// TIA Portal V17 export
// export: Created 2024-09-02T12:50:19.8771869Z, ExportSetting WithDefaults, DisplayName Totally Integrated Automation Portal, DisplayVersion V17, DisplayName TIA Portal Openness, DisplayVersion V17, DisplayName TIA Portal Version Control Interface, DisplayVersion V17, DisplayName STEP 7 Professional, DisplayVersion V17, DisplayName STEP 7 Safety, DisplayVersion V17, DisplayName WinCC Professional, DisplayVersion V17
FUNCTION "AnwFC1_FG02_Parameter_SLG3_OP70" : Void   // FC1111, LAD
TITLE = Parameter Moby / Parameter Moby
{ S7_Optimized_Access := 'TRUE' }
AUTHOR : OlegFuehrus
FAMILY : MOBY
NAME : OlegFuehrus
VERSION : 0.1
// stored: AutoNumber false, IsIECCheckEnabled false, SetENOAutomatically false, UDAEnableTagReadback false
   VAR_TEMP
      Motion_Release : Bool;
      Hand : Bool;
      Auto : Bool;
      t_VKE0 : Bool;
      t_VKE1 : Bool;
      t_reset : Bool;
      t_read : Bool;
      t_read_ok : Bool;
      t_write : Bool;
      t_write_ok : Bool;
      t_TAFmaske : Byte;
      t_PageNr_Station : Int;
      t_PageNr_Station_Before : Int;
      t_Nr : Int;
      Length_of_Db : Int;
   END_VAR
   VAR_TEMP   // added for the SCL form of the ladder/FBD networks
      _w1 : Bool;
   END_VAR
BEGIN

REGION Network 1: VKE 0/1
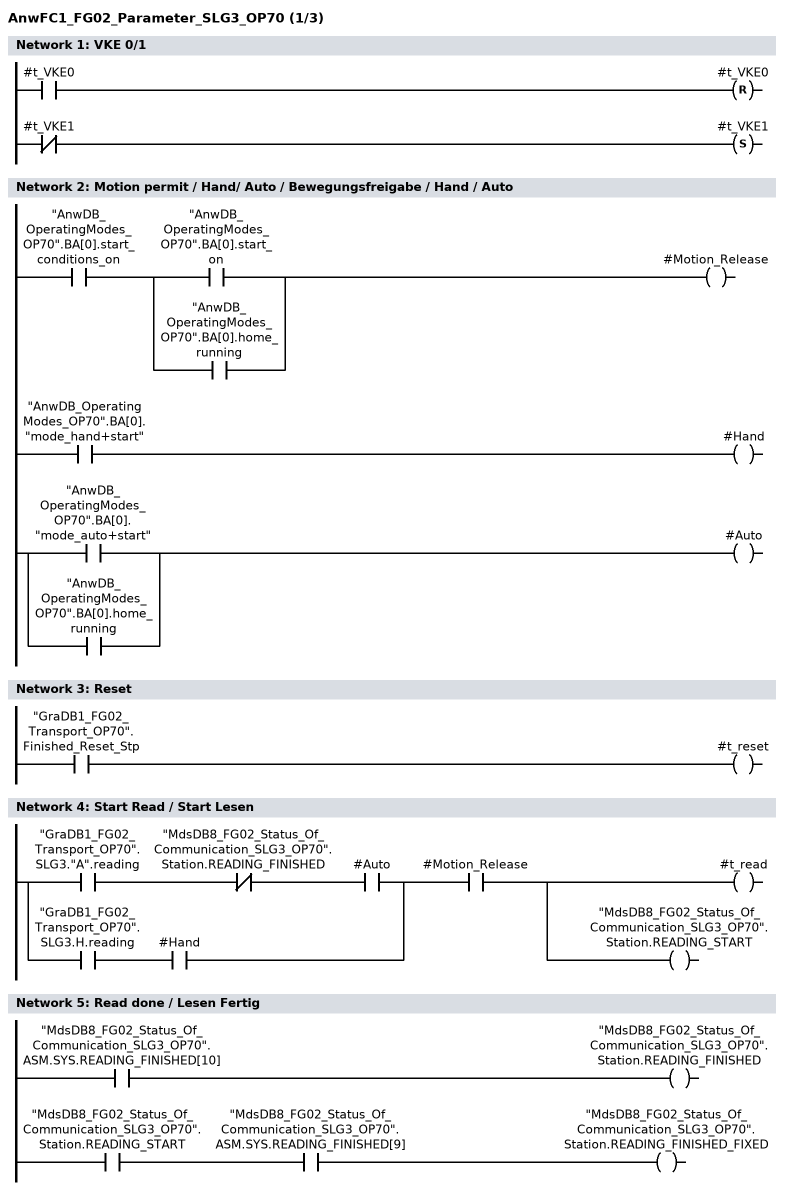
   RUNG wire#powerrail
      Contact( #t_VKE0 )
      R_Coil( #t_VKE0 )
   END_RUNG
   RUNG wire#powerrail
      I_Contact( #t_VKE1 )
      S_Coil( #t_VKE1 )
   END_RUNG
   // the same network as SCL:
   IF #t_VKE0 THEN #t_VKE0 := FALSE; END_IF;
   IF NOT #t_VKE1 THEN #t_VKE1 := TRUE; END_IF;
END_REGION

REGION Network 2: Motion permit / Hand/ Auto / Bewegungsfreigabe / Hand / Auto
   RUNG wire#powerrail
      Contact( "AnwDB_OperatingModes_OP70".BA[0].start_conditions_on )
      wire#w1
      Contact( "AnwDB_OperatingModes_OP70".BA[0].start_on )
      wire#w2
      Coil( #Motion_Release )
   END_RUNG
   RUNG wire#w1
      Contact( "AnwDB_OperatingModes_OP70".BA[0].home_running )
   END_RUNG wire#w2
   RUNG wire#powerrail
      Contact( "AnwDB_OperatingModes_OP70".BA[0]."mode_hand+start" )
      Coil( #Hand )
   END_RUNG
   RUNG wire#powerrail
      Contact( "AnwDB_OperatingModes_OP70".BA[0]."mode_auto+start" )
      wire#w3
      Coil( #Auto )
   END_RUNG
   RUNG wire#powerrail
      Contact( "AnwDB_OperatingModes_OP70".BA[0].home_running )
   END_RUNG wire#w3
   // the same network as SCL:
   #Motion_Release := "AnwDB_OperatingModes_OP70".BA[0].start_conditions_on AND ("AnwDB_OperatingModes_OP70".BA[0].start_on OR "AnwDB_OperatingModes_OP70".BA[0].home_running);
   #Hand := "AnwDB_OperatingModes_OP70".BA[0]."mode_hand+start";
   #Auto := "AnwDB_OperatingModes_OP70".BA[0]."mode_auto+start" OR "AnwDB_OperatingModes_OP70".BA[0].home_running;
END_REGION

REGION Network 3: Reset
   RUNG wire#powerrail
      Contact( "GraDB1_FG02_Transport_OP70".Finished_Reset_Stp )
      Coil( #t_reset )
   END_RUNG
   // the same network as SCL:
   #t_reset := "GraDB1_FG02_Transport_OP70".Finished_Reset_Stp;
END_REGION

REGION Network 4: Start Read / Start Lesen
   RUNG wire#powerrail
      Contact( "GraDB1_FG02_Transport_OP70".SLG3."A".reading )
      I_Contact( "MdsDB8_FG02_Status_Of_Communication_SLG3_OP70".Station.READING_FINISHED )
      Contact( #Auto )
      wire#w1
      Contact( #Motion_Release )
      wire#w2
      Coil( #t_read )
   END_RUNG
   RUNG wire#powerrail
      Contact( "GraDB1_FG02_Transport_OP70".SLG3.H.reading )
      Contact( #Hand )
   END_RUNG wire#w1
   RUNG wire#w2
      Coil( "MdsDB8_FG02_Status_Of_Communication_SLG3_OP70".Station.READING_START )
   END_RUNG
   // the same network as SCL:
   #t_read := (("GraDB1_FG02_Transport_OP70".SLG3."A".reading AND NOT "MdsDB8_FG02_Status_Of_Communication_SLG3_OP70".Station.READING_FINISHED AND #Auto) OR ("GraDB1_FG02_Transport_OP70".SLG3.H.reading AND #Hand)) AND #Motion_Release;
   "MdsDB8_FG02_Status_Of_Communication_SLG3_OP70".Station.READING_START := #t_read;
END_REGION

REGION Network 5: Read done / Lesen Fertig
   RUNG wire#powerrail
      Contact( "MdsDB8_FG02_Status_Of_Communication_SLG3_OP70".ASM.SYS.READING_FINISHED[10] )
      Coil( "MdsDB8_FG02_Status_Of_Communication_SLG3_OP70".Station.READING_FINISHED )
   END_RUNG
   RUNG wire#powerrail
      Contact( "MdsDB8_FG02_Status_Of_Communication_SLG3_OP70".Station.READING_START )
      Contact( "MdsDB8_FG02_Status_Of_Communication_SLG3_OP70".ASM.SYS.READING_FINISHED[9] )
      Coil( "MdsDB8_FG02_Status_Of_Communication_SLG3_OP70".Station.READING_FINISHED_FIXED )
   END_RUNG
   // the same network as SCL:
   "MdsDB8_FG02_Status_Of_Communication_SLG3_OP70".Station.READING_FINISHED := "MdsDB8_FG02_Status_Of_Communication_SLG3_OP70".ASM.SYS.READING_FINISHED[10];
   "MdsDB8_FG02_Status_Of_Communication_SLG3_OP70".Station.READING_FINISHED_FIXED := "MdsDB8_FG02_Status_Of_Communication_SLG3_OP70".Station.READING_START AND "MdsDB8_FG02_Status_Of_Communication_SLG3_OP70".ASM.SYS.READING_FINISHED[9];
END_REGION

REGION Network 6: Start Writing / Start Schreiben
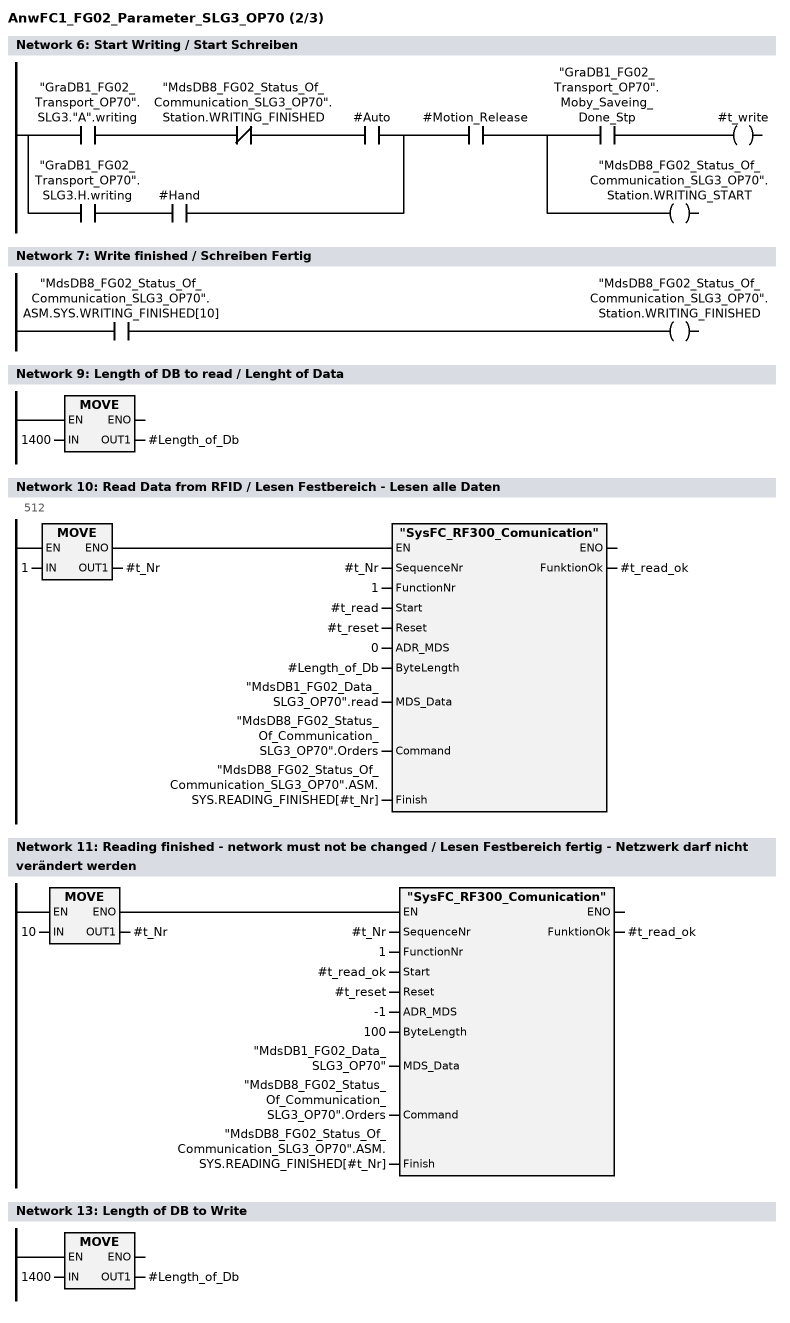
   RUNG wire#powerrail
      Contact( "GraDB1_FG02_Transport_OP70".SLG3."A".writing )
      I_Contact( "MdsDB8_FG02_Status_Of_Communication_SLG3_OP70".Station.WRITING_FINISHED )
      Contact( #Auto )
      wire#w1
      Contact( #Motion_Release )
      wire#w2
      Contact( "GraDB1_FG02_Transport_OP70".Moby_Saveing_Done_Stp )
      Coil( #t_write )
   END_RUNG
   RUNG wire#powerrail
      Contact( "GraDB1_FG02_Transport_OP70".SLG3.H.writing )
      Contact( #Hand )
   END_RUNG wire#w1
   RUNG wire#w2
      Coil( "MdsDB8_FG02_Status_Of_Communication_SLG3_OP70".Station.WRITING_START )
   END_RUNG
   // the same network as SCL:
   #_w1 := (("GraDB1_FG02_Transport_OP70".SLG3."A".writing AND NOT "MdsDB8_FG02_Status_Of_Communication_SLG3_OP70".Station.WRITING_FINISHED AND #Auto) OR ("GraDB1_FG02_Transport_OP70".SLG3.H.writing AND #Hand)) AND #Motion_Release;
   #t_write := #_w1 AND "GraDB1_FG02_Transport_OP70".Moby_Saveing_Done_Stp;
   "MdsDB8_FG02_Status_Of_Communication_SLG3_OP70".Station.WRITING_START := #_w1;
END_REGION

REGION Network 7: Write finished / Schreiben Fertig
   RUNG wire#powerrail
      Contact( "MdsDB8_FG02_Status_Of_Communication_SLG3_OP70".ASM.SYS.WRITING_FINISHED[10] )
      Coil( "MdsDB8_FG02_Status_Of_Communication_SLG3_OP70".Station.WRITING_FINISHED )
   END_RUNG
   // the same network as SCL:
   "MdsDB8_FG02_Status_Of_Communication_SLG3_OP70".Station.WRITING_FINISHED := "MdsDB8_FG02_Status_Of_Communication_SLG3_OP70".ASM.SYS.WRITING_FINISHED[10];
END_REGION

REGION Network 8: ######## READ PARAMETER ########
END_REGION

REGION Network 9: Length of DB to read / Lenght of Data
   RUNG wire#powerrail
      Move(in := 1400, out1 => #Length_of_Db)
   END_RUNG
   // the same network as SCL:
   #Length_of_Db := 1400;
END_REGION

REGION Network 10: Read Data from RFID / Lesen Festbereich - Lesen alle Daten
   // 512
   RUNG wire#powerrail
      Move(in := 1, out1 => #t_Nr)
      "SysFC_RF300_Comunication"(SequenceNr := #t_Nr, FunctionNr := 1, Start := #t_read, Reset := #t_reset, ADR_MDS := 0, ByteLength := #Length_of_Db, MDS_Data := "MdsDB1_FG02_Data_SLG3_OP70".read, Command := "MdsDB8_FG02_Status_Of_Communication_SLG3_OP70".Orders, Finish := "MdsDB8_FG02_Status_Of_Communication_SLG3_OP70".ASM.SYS.READING_FINISHED[#t_Nr], FunktionOk => #t_read_ok)
   END_RUNG
   // the same network as SCL:
   #t_Nr := 1;
   "SysFC_RF300_Comunication"(SequenceNr := #t_Nr,
                           FunctionNr := 1,
                           Start := #t_read,
                           Reset := #t_reset,
                           ADR_MDS := 0,
                           ByteLength := #Length_of_Db,
                           MDS_Data := "MdsDB1_FG02_Data_SLG3_OP70".read,
                           Command := "MdsDB8_FG02_Status_Of_Communication_SLG3_OP70".Orders,
                           Finish := "MdsDB8_FG02_Status_Of_Communication_SLG3_OP70".ASM.SYS.READING_FINISHED[#t_Nr],
                           FunktionOk => #t_read_ok);
END_REGION

REGION Network 11: Reading finished - network must not be changed / Lesen Festbereich fertig - Netzwerk darf nicht verändert werden
   RUNG wire#powerrail
      Move(in := 10, out1 => #t_Nr)
      "SysFC_RF300_Comunication"(SequenceNr := #t_Nr, FunctionNr := 1, Start := #t_read_ok, Reset := #t_reset, ADR_MDS := -1, ByteLength := 100, MDS_Data := "MdsDB1_FG02_Data_SLG3_OP70", Command := "MdsDB8_FG02_Status_Of_Communication_SLG3_OP70".Orders, Finish := "MdsDB8_FG02_Status_Of_Communication_SLG3_OP70".ASM.SYS.READING_FINISHED[#t_Nr], FunktionOk => #t_read_ok)
   END_RUNG
   // the same network as SCL:
   #t_Nr := 10;
   "SysFC_RF300_Comunication"(SequenceNr := #t_Nr,
                           FunctionNr := 1,
                           Start := #t_read_ok,
                           Reset := #t_reset,
                           ADR_MDS := -1,
                           ByteLength := 100,
                           MDS_Data := "MdsDB1_FG02_Data_SLG3_OP70",
                           Command := "MdsDB8_FG02_Status_Of_Communication_SLG3_OP70".Orders,
                           Finish := "MdsDB8_FG02_Status_Of_Communication_SLG3_OP70".ASM.SYS.READING_FINISHED[#t_Nr],
                           FunktionOk => #t_read_ok);
END_REGION

REGION Network 12: ######## WRITE PARAMETER ########
END_REGION

REGION Network 13: Length of DB to Write
   RUNG wire#powerrail
      Move(in := 1400, out1 => #Length_of_Db)
   END_RUNG
   // the same network as SCL:
   #Length_of_Db := 1400;
END_REGION

REGION Network 14: Write - whole data to RFID / Schreiben - komplett
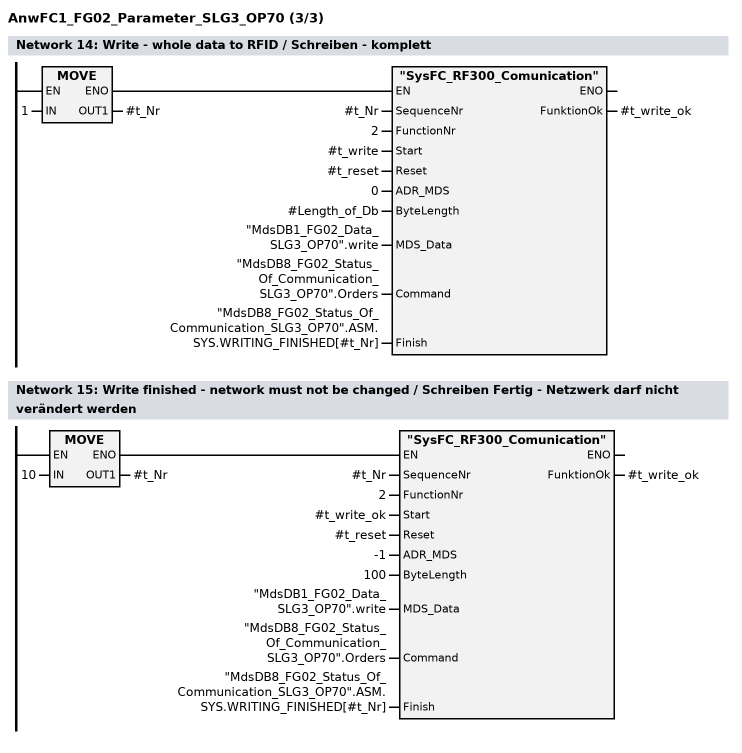
   RUNG wire#powerrail
      Move(in := 1, out1 => #t_Nr)
      "SysFC_RF300_Comunication"(SequenceNr := #t_Nr, FunctionNr := 2, Start := #t_write, Reset := #t_reset, ADR_MDS := 0, ByteLength := #Length_of_Db, MDS_Data := "MdsDB1_FG02_Data_SLG3_OP70".write, Command := "MdsDB8_FG02_Status_Of_Communication_SLG3_OP70".Orders, Finish := "MdsDB8_FG02_Status_Of_Communication_SLG3_OP70".ASM.SYS.WRITING_FINISHED[#t_Nr], FunktionOk => #t_write_ok)
   END_RUNG
   // the same network as SCL:
   #t_Nr := 1;
   "SysFC_RF300_Comunication"(SequenceNr := #t_Nr,
                           FunctionNr := 2,
                           Start := #t_write,
                           Reset := #t_reset,
                           ADR_MDS := 0,
                           ByteLength := #Length_of_Db,
                           MDS_Data := "MdsDB1_FG02_Data_SLG3_OP70".write,
                           Command := "MdsDB8_FG02_Status_Of_Communication_SLG3_OP70".Orders,
                           Finish := "MdsDB8_FG02_Status_Of_Communication_SLG3_OP70".ASM.SYS.WRITING_FINISHED[#t_Nr],
                           FunktionOk => #t_write_ok);
END_REGION

REGION Network 15: Write finished - network must not be changed / Schreiben Fertig - Netzwerk darf nicht verändert werden
   RUNG wire#powerrail
      Move(in := 10, out1 => #t_Nr)
      "SysFC_RF300_Comunication"(SequenceNr := #t_Nr, FunctionNr := 2, Start := #t_write_ok, Reset := #t_reset, ADR_MDS := -1, ByteLength := 100, MDS_Data := "MdsDB1_FG02_Data_SLG3_OP70".write, Command := "MdsDB8_FG02_Status_Of_Communication_SLG3_OP70".Orders, Finish := "MdsDB8_FG02_Status_Of_Communication_SLG3_OP70".ASM.SYS.WRITING_FINISHED[#t_Nr], FunktionOk => #t_write_ok)
   END_RUNG
   // the same network as SCL:
   #t_Nr := 10;
   "SysFC_RF300_Comunication"(SequenceNr := #t_Nr,
                           FunctionNr := 2,
                           Start := #t_write_ok,
                           Reset := #t_reset,
                           ADR_MDS := -1,
                           ByteLength := 100,
                           MDS_Data := "MdsDB1_FG02_Data_SLG3_OP70".write,
                           Command := "MdsDB8_FG02_Status_Of_Communication_SLG3_OP70".Orders,
                           Finish := "MdsDB8_FG02_Status_Of_Communication_SLG3_OP70".ASM.SYS.WRITING_FINISHED[#t_Nr],
                           FunktionOk => #t_write_ok);
END_REGION

REGION Network 16: #############################
END_REGION
END_FUNCTION
